// TIA Portal V18 export
FUNCTION_BLOCK "FC51_Control"   // FB4, FBD
{ S7_Optimized_Access := 'TRUE' }
// stored: MemoryReserve 100, SetENOAutomatically false
   VAR_INPUT
      I_Start : Bool;   // 固定速度启动
      I_Frequency : Real;
      I_Alarm_Confirm : Bool;
   END_VAR
   VAR
      FB_Always_True : Bool;
      Frequency_Trans_Instance { ExternalAccessible := 'False'; ExternalVisible := 'False'; ExternalWritable := 'False'} : "Frequency_Trans";
      FC51_Modbus_Com_Instance { S7_SetPoint := 'True'} : "FC51_Modbus_Com";
   END_VAR
   VAR_TEMP   // added for the SCL form of the ladder/FBD networks
      _w1 : Bool;
   END_VAR
BEGIN

REGION Network 1
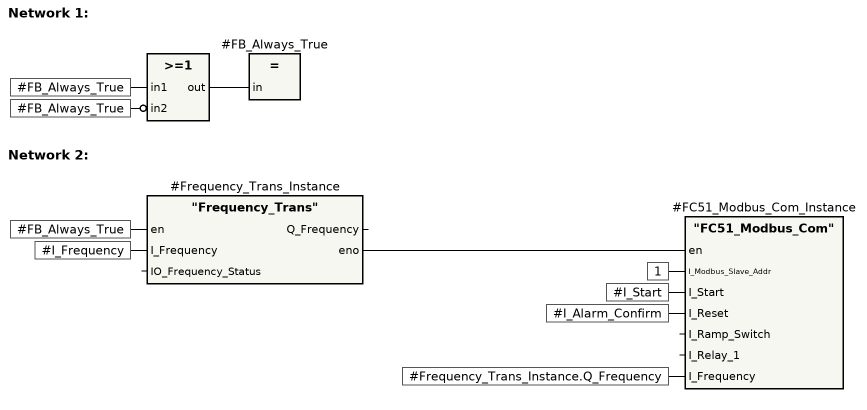
   #FB_Always_True := #FB_Always_True OR NOT #FB_Always_True;
END_REGION

REGION Network 2
   #Frequency_Trans_Instance(EN := #FB_Always_True, I_Frequency := #I_Frequency, ENO => #_w1);   // "Frequency_Trans"
   IF #_w1 THEN
       #FC51_Modbus_Com_Instance(I_Modbus_Slave_Addr := 1,   // "FC51_Modbus_Com"
                               I_Start := #I_Start,
                               I_Reset := #I_Alarm_Confirm,
                               I_Frequency := #Frequency_Trans_Instance.Q_Frequency);
   END_IF;
END_REGION
END_FUNCTION_BLOCK
